Staubli VAL3: stopCycle.pgx

program stopCycle()
begin
  //
  // STOP
  //
  stopMove()
  cycleStatus:bToStop=true
  call use:timerDialog(" STOP CYCLE ",1)
  //
  watch(cycleStatus:bToStop==false,1)
end
